Staubli VAL3: selectPath.pgx

program selectPath()
  local num l_nKey
  local num l_nSelected
begin
  //
  nPage=2
  bUserRefresh=bListRefresh=true
  sNewPath=""
  l_nSelected=nSelected
  do
    call Refresh()
    call RefreshList()
    call user:setList("路径",sList,bUserRefresh,bListRefresh,nSelected,sItem,l_nKey)
    bUserRefresh=false
    bListRefresh=false
    call MainKey(l_nKey)
    delay(0)
  until bExit
  //
  if sPathList[l_nSelected]!=""
    if sNewPath!=""
      insert(sPathList[l_nSelected+1])
      sPathList[l_nSelected+1]=sNewPath
    endIf
  else
    sPathList[l_nSelected]=sNewPath
  endIf

  nPage=1
  bUserRefresh=bListRefresh=true
  bExit=false
end
